
// ===== library types =====

TYPE "UDT_Node_INT_G2"
   STRUCT
      Enable : Bool := FALSE;   // Enable polling for this slave node (TRUE = Active)
      SlaveAddress : UInt := 1;   // Modbus RTU slave address (1..247)
      SwapWords : Bool := FALSE;
      Requests : Array[1..10] of "UDT_Request_INT_G2";   // Data Address Of Slave Device
   END_STRUCT;
END_TYPE

TYPE "UDT_Request_INT_G2"
   STRUCT
      Enable : Bool := FALSE;   // Enable or disable this specific request (TRUE = Active)
      Mode : USInt := 1;   // Modbus function mode (0: Read, 1: Write)
      DataAddress : UDInt := 40001;   // Modbus register start address (e.g., 40001, 30001)
      DataLen : UInt := 1;   // Number of registers to read/write (Max 10 )
      IsDouble : Bool := FALSE;   // False = 16-bit, True = 32-bit
      DataValue : Array[0..9] of DInt;   // Data value to write to slave or value received from slave
      Done : Bool := FALSE;   // Execution status (TRUE = Request completed successfully)
      Error : Bool := FALSE;   // Execution status (TRUE = Request failed or timed out)
      Status : Word := 16#0;   // Modbus status code / error code from MB_MASTER
   END_STRUCT;
END_TYPE